// Mitsubishi GX Works2 project: BIN_CLL_502_100_Z001_Demo   PLC: Q04UDEH

TYPE DUT_BNI_CCL_502_100_Z001_P1_5_Rx : STRUCT
  Port0_In0 : BOOL;
  Port0_In1 : BOOL;
  Port1_In2 : BOOL;
  Port1_In3 : BOOL;
  Port2_In4 : BOOL;
  Port2_In5 : BOOL;
  Port3_In6 : BOOL;
  Port3_In7 : BOOL;
  Port4_In8 : BOOL;
  Port4_In9 : BOOL;
  Port5_InA : BOOL;
  Port5_InB : BOOL;
  Port6_InC : BOOL;
  Port6_InD : BOOL;
  Port7_InE : BOOL;
  Port7_InF : BOOL;
  Port0_InOut0_Diagnostic : BOOL;
  Port0_InOut1_Diagnostic : BOOL;
  Port1_InOut2_Diagnostic : BOOL;
  Port1_InOut3_Diagnostic : BOOL;
  Port2_InOut4_Diagnostic : BOOL;
  Port2_InOut5_Diagnostic : BOOL;
  Port3_InOut6_Diagnostic : BOOL;
  Port3_InOut7_Diagnostic : BOOL;
  Port4_InOut8_Diagnostic : BOOL;
  Port4_InOut9_Diagnostic : BOOL;
  Port5_InOutA_Diagnostic : BOOL;
  Port5_InOutB_Diagnostic : BOOL;
  Port6_InOutC_Diagnostic : BOOL;
  Port6_InOutD_Diagnostic : BOOL;
  Port7_InOutE_Diagnostic : BOOL;
  Port7_InOutF_Diagnostic : BOOL;
  Port0_Diagnostic : BOOL;
  Port1_Diagnostic : BOOL;
  Port2_Diagnostic : BOOL;
  Port3_Diagnostic : BOOL;
  Port4_Diagnostic : BOOL;
  Port5_Diagnostic : BOOL;
  Port6_Diagnostic : BOOL;
  Port7_Diagnostic : BOOL;
  Us_UnderVoltage : BOOL;
  Ua_UnderVlotage : BOOL;
  bRx_x2A : BOOL;
  bRx_x2B : BOOL;
  bRx_x2C : BOOL;
  bRx_x2D : BOOL;
  bRx_x2E : BOOL;
  bRx_x2F : BOOL;
  IOLINK_Ch0_Established : BOOL;
  IOLINK_Ch1_Established : BOOL;
  IOLINK_Ch2_Established : BOOL;
  IOLINK_Ch3_Established : BOOL;
  bRx_x34 : BOOL;
  bRx_x35 : BOOL;
  bRx_x36 : BOOL;
  bRx_x37 : BOOL;
  IOLINK_Ch0_EventFlag : BOOL;
  IOLINK_Ch1_EventFlag : BOOL;
  IOLINK_Ch2_EventFlag : BOOL;
  IOLINK_Ch3_EventFlag : BOOL;
  bRx_x3C : BOOL;
  bRx_x3D : BOOL;
  bRx_x3E : BOOL;
  bRx_x3F : BOOL;
  IOLINK_Ch0_DataValid : BOOL;
  IOLINK_Ch1_DataValid : BOOL;
  IOLINK_Ch2_DataValid : BOOL;
  IOLINK_Ch3_DataValid : BOOL;
  bRx_x44 : BOOL;
  bRx_x45 : BOOL;
  bRx_x46 : BOOL;
  bRx_x47 : BOOL;
  bRx_x48 : BOOL;
  bRx_x49 : BOOL;
  bRx_x4A : BOOL;
  bRx_x4B : BOOL;
  bRx_x4C : BOOL;
  bRx_x4D : BOOL;
  bRx_x4E : BOOL;
  bRx_x4F : BOOL;
END_STRUCT END_TYPE

TYPE DUT_BNI_CCL_502_100_Z001_P1_5_Ry : STRUCT
  Port0_Out0 : BOOL;
  Port0_Out1 : BOOL;
  Port1_Out2 : BOOL;
  Port1_Out3 : BOOL;
  Port2_Out4 : BOOL;
  Port2_Out5 : BOOL;
  Port3_Out6 : BOOL;
  Port3_Out7 : BOOL;
  Port4_Out8 : BOOL;
  Port4_Out9 : BOOL;
  Port5_OutA : BOOL;
  Port5_OutB : BOOL;
  Port6_OutC : BOOL;
  Port6_OutD : BOOL;
  Port7_OutE : BOOL;
  Port7_OutF : BOOL;
  Port0_IsOutput : BOOL;
  Port1_IsOutput : BOOL;
  Port2_IsOutput : BOOL;
  Port3_IsOutput : BOOL;
  Port4_IsOutput : BOOL;
  Port5_IsOutput : BOOL;
  Port6_IsOutput : BOOL;
  Port7_IsOutput : BOOL;
  Port8_IsOutput : BOOL;
  Port9_IsOutput : BOOL;
  PortA_IsOutput : BOOL;
  PortB_IsOutput : BOOL;
  PortC_IsOutput : BOOL;
  PortD_IsOutput : BOOL;
  PortE_IsOutput : BOOL;
  PortF_IsOutput : BOOL;
  Display_LED_Red : BOOL;
  Display_LED_Green : BOOL;
  Display_LOCK : BOOL;
  bRY_x23 : BOOL;
  bRY_x24 : BOOL;
  bRY_x25 : BOOL;
  bRY_x26 : BOOL;
  bRY_x27 : BOOL;
  bRY_x28 : BOOL;
  bRY_x2A : BOOL;
  bRY_x2B : BOOL;
  bRY_x2C : BOOL;
  bRY_x2D : BOOL;
  bRY_x2E : BOOL;
  bRY_x2F : BOOL;
  bRY_x29 : BOOL;
  IOLINK_Ch0_Enable : BOOL;
  IOLINK_Ch1_Enable : BOOL;
  IOLINK_Ch2_Enable : BOOL;
  IOLINK_Ch3_Enable : BOOL;
  bRY_x34 : BOOL;
  bRY_x35 : BOOL;
  bRY_x36 : BOOL;
  bRY_x37 : BOOL;
  IOLINK_Ch0_EventClear : BOOL;
  IOLINK_Ch1_EventClear : BOOL;
  IOLINK_Ch2_EventClear : BOOL;
  IOLINK_Ch3_EventClear : BOOL;
  bRY_x3C : BOOL;
  bRY_x3D : BOOL;
  bRY_x3E : BOOL;
  bRY_x3F : BOOL;
  bRY_x40 : BOOL;
  bRY_x41 : BOOL;
  bRY_x42 : BOOL;
  bRY_x43 : BOOL;
  bRY_x44 : BOOL;
  bRY_x45 : BOOL;
  bRY_x46 : BOOL;
  bRY_x47 : BOOL;
  bRY_x48 : BOOL;
  bRY_x49 : BOOL;
  bRY_x4A : BOOL;
  bRY_x4B : BOOL;
  bRY_x4C : BOOL;
  bRY_x4D : BOOL;
  bRY_x4E : BOOL;
  bRY_x4F : BOOL;
END_STRUCT END_TYPE

TYPE D_QJ61BT11N_IN : STRUCT
  x0ModuleError : BOOL;  (* This signal indicates whether the module is normal or faulty,True=Error *)
  x1HostDataOK : BOOL;  (* This signal indicates the data link status of the host station,True=Data Link in Process *)
  x2NotUsed : BOOL;
  x3OtherStLink : BOOL;  (* This signal indicates the data link status of other stations,True= Have Fautly Station *)
  x4NotUsed : BOOL;
  x5NotUsed : BOOL;
  x6NotUsed : BOOL;
  x7NotUsed : BOOL;
  x8NotUsed : BOOL;
  x9NotUsed : BOOL;
  xANotUsed : BOOL;
  xBNotUsed : BOOL;
  xCNotUsed : BOOL;
  xDNotUsed : BOOL;
  xENotUsed : BOOL;
  xFReady : BOOL;  (* This signal indicates whether the module is ready to operate,True=Ready *)
  x10NotUsed : BOOL;
  x11NotUsed : BOOL;
  x12NotUsed : BOOL;
  x13NotUsed : BOOL;
  x14NotUsed : BOOL;
  x15NotUsed : BOOL;
  x16NotUsed : BOOL;
  x17NotUsed : BOOL;
  x18NotUsed : BOOL;
  x19NotUsed : BOOL;
  x1ANotUsed : BOOL;
  x1BNotUsed : BOOL;
  x1CNotUsed : BOOL;
  x1DNotUsed : BOOL;
  x1ENotUsed : BOOL;
  x1FNotUsed : BOOL;
END_STRUCT END_TYPE

TYPE DUT_BNI_CCL_502_100_Z001_Ry3 : STRUCT
  bRy_mn0 : BOOL;
  bRy_mn1 : BOOL;
  bRy_mn2 : BOOL;
  bRy_mn3 : BOOL;
  bRy_mn4 : BOOL;
  bRy_mn5 : BOOL;
  bRy_mn6 : BOOL;
  bRy_mn7 : BOOL;
  InitDataProcessing : BOOL;
  InitDataRequest : BOOL;
  ErrorResetRequest : BOOL;
  bRy_mnB : BOOL;
  MessageTransferReq : BOOL;
  MessageTransferHandShake : BOOL;
  bRy_mnE : BOOL;
  bRy_mnF : BOOL;
END_STRUCT END_TYPE

TYPE DUT_BNI_CCL_502_100_Z001_Rx3 : STRUCT
  bRx_mn0 : BOOL;
  bRx_mn1 : BOOL;
  bRx_mn2 : BOOL;
  bRx_mn3 : BOOL;
  MessageSize0 : BOOL;
  MessageSize1 : BOOL;
  MessageSize2 : BOOL;
  bRx_mn7 : BOOL;
  InitDataProcessing : BOOL;
  InitDataComplete : BOOL;
  ErrorStautsFlag : BOOL;
  RemoteReady : BOOL;
  MessageTransferAccept : BOOL;
  MessageTransferHandShake : BOOL;
  bRx_mnE : BOOL;
  bRx_mnF : BOOL;
END_STRUCT END_TYPE

TYPE DUT_BNI_CCL_502_100_Z001_P5_Rwr : STRUCT
  IOLINK_Ch0 : ARRAY [0..15] OF INT;
  IOLINK_Ch1 : ARRAY [0..15] OF INT;
  IOLINK_Ch2 : ARRAY [0..15] OF INT;
  IOLINK_Ch3 : ARRAY [0..15] OF INT;
END_STRUCT END_TYPE

TYPE DUT_BNI_CCL_502_100_Z001_P5_Rww : STRUCT
  IOLINK_Ch0 : ARRAY [0..15] OF INT;
  IOLINK_Ch1 : ARRAY [0..15] OF INT;
  IOLINK_Ch2 : ARRAY [0..15] OF INT;
  IOLINK_Ch3 : ARRAY [0..15] OF INT;
END_STRUCT END_TYPE

// global labels: Global1
VAR_GLOBAL
  CCLINK_Module1 : D_QJ61BT11N_IN;
  BNI_CCL_502_Z001_1_Ry3 : DUT_BNI_CCL_502_100_Z001_Ry3;
  BNI_CCL_502_Z001_1_Rx3 : DUT_BNI_CCL_502_100_Z001_Rx3;
  BNI_CCL_502_Z001_1_Rx0 : DUT_BNI_CCL_502_100_Z001_P1_5_Rx;
  BNI_CCL_502_Z001_1_Ry0 : DUT_BNI_CCL_502_100_Z001_P1_5_Ry;
  BNI_CCL_502_Z001_1_Rwr : DUT_BNI_CCL_502_100_Z001_P5_Rwr;
  BNI_CCL_502_Z001_1_Rww : DUT_BNI_CCL_502_100_Z001_P5_Rww;
END_VAR

// task Task_01 (event TRUE, interval 0, priority 31): POU_01

PROGRAM POU_01
VAR
  HandShake : FB_BNI_CCL_502_Z001_HandShake;
  bConfig : BOOL;
  RWM1 : FB_CONTRINEX;
END_VAR

IF NOT bConfig THEN
	BNI_CCL_502_Z001_1_Ry0.Port0_IsOutput:=TRUE;
	BNI_CCL_502_Z001_1_Ry0.Port1_IsOutput:=TRUE;
	BNI_CCL_502_Z001_1_Ry0.IOLINK_Ch0_Enable:=TRUE;
	BNI_CCL_502_Z001_1_Ry0.IOLINK_Ch1_Enable:=TRUE;
	BNI_CCL_502_Z001_1_Ry0.IOLINK_Ch2_Enable:=TRUE;
	BNI_CCL_502_Z001_1_Ry0.IOLINK_Ch3_Enable:=TRUE;
	bConfig:=TRUE;
END_IF;


RWM1(	
	IOLINKData:=BNI_CCL_502_Z001_1_Rwr.IOLINK_Ch2
	,HaveTags:=M0
	,NBTags:=D10
	,UID0:=D11
	,UID1:=D12
	,UID2:=D13
	,UID3:=D14
	,UID4:=D15
	,UID5:=D16
	,UID6:=D17
	,UID7:=D18
	);


HandShake(
	Rx3:=BNI_CCL_502_Z001_1_Rx3
	,bConfig:=bConfig
	,bCCLinkMasterStatus:=CCLINK_Module1.xFReady
	,Ry3:=BNI_CCL_502_Z001_1_Ry3
	);
END_PROGRAM

FUNCTION_BLOCK FB_BNI_CCL_502_Z001_HandShake
VAR_INPUT
  Rx3 : DUT_BNI_CCL_502_100_Z001_Rx3;
END_VAR
VAR_OUTPUT
  Ry3 : DUT_BNI_CCL_502_100_Z001_Ry3;
END_VAR
VAR
  iStep : INT;
END_VAR
VAR_INPUT
  bInitIO : BOOL;
  bCCLinkMasterStatus : BOOL;
END_VAR
VAR_OUTPUT
  bRemoteOK : BOOL;
END_VAR
VAR_INPUT
  bConfig : BOOL;
END_VAR


(*Auto Reset*)
	Ry3.ErrorResetRequest:=Rx3.ErrorStautsFlag AND bCCLinkMasterStatus;

(*Data Initing..*)	
 	Ry3.InitDataProcessing:=Rx3.InitDataProcessing AND bCCLinkMasterStatus AND bConfig;

(*Remote OK*)
	bRemoteOK:=Rx3.RemoteReady;
END_FUNCTION_BLOCK

FUNCTION_BLOCK FB_CONTRINEX
VAR_INPUT
  IOLINKData : ARRAY [0..15] OF INT;
END_VAR
VAR_OUTPUT
  HaveTags : BOOL;
  RFField : BOOL;
  NBTags : WORD;
  UID0 : WORD;
  UID1 : WORD;
  UID2 : WORD;
  UID3 : WORD;
  UID4 : WORD;
  UID5 : WORD;
  UID6 : WORD;
  UID7 : WORD;
END_VAR


D0:=IOLINKData[0];

RFField:= (D0&2#0001_0000_0000_0000) <> 0 ;
HaveTags:= (D0&2#0010_0000_0000_0000) <> 0 ;

NBTags:= SHR((D0&2#0000_1111_0000_0000),8);

UID0:=D0&2#0000_0000_1111_1111;

D0:=IOLINKData[1];
UID1:=SHR((D0&2#1111_1111_0000_0000),8);
UID2:=SHR((D0&2#0000_0000_1111_1111),8);

D0:=IOLINKData[2];
UID3:=SHR((D0&2#1111_1111_0000_0000),8);
UID4:=SHR((D0&2#0000_0000_1111_1111),8);

D0:=IOLINKData[3];
UID5:=SHR((D0&2#1111_1111_0000_0000),8);
UID6:=SHR((D0&2#0000_0000_1111_1111),8);

D0:=IOLINKData[4];
UID5:=SHR((D0&2#1111_1111_0000_0000),8);

;
END_FUNCTION_BLOCK
